FUNCTION_BLOCK XboxController
VAR_INPUT
END_VAR
VAR_OUTPUT
	
			XboxController				: 		FB_Xbox_Controller(NetID := '', iControllerNumber := 1);
			bIsConnected   				:  		ARRAY [1..2] OF BOOL;

			Start 						:       BOOL; 
			Reset 						:       BOOL;
			Button_A            		:       BOOL;
			Button_B                 	:       BOOL;
			Button_X             		:       BOOL;
			Button_Y                    :       BOOL;
			Dpad_U	                    :       BOOL;
			Dpad_D	                    :       BOOL;
			lBumper	                    :       BOOL;
			rBumper	                    :       BOOL;
			lTrigger                    :       LREAL;
			rTrigger                    :       LREAL;
			lStick_Y	                :       LREAL;
			lStick_X	                :       LREAL;
     		rStick_Y	                :       LREAL;
     		rStick_X	                :       LREAL;
			
END_VAR
VAR    
END_VAR

Cyclic();

METHOD clearScreenshot : BOOL
VAR_INPUT
	
bDpad_U 					: BOOL; 

END_VAR
END_METHOD

ACTION Cyclic:
XboxController.Cycle();
mapping(); 
init();
bIsConnected[1] := XboxController.P_Status.bConnected;
END_ACTION

METHOD Init
VAR_INPUT
END_VAR
END_METHOD

ACTION Mapping:




// Button Mapping
Start 				:= XboxController.P_Buttons.bStart;
Reset 				:= XboxController.P_Buttons.bBack;
Button_A 			:= XboxController.P_Buttons.bA_Button;
Button_B 			:= XboxController.P_Buttons.bB_Button;
Button_X 			:= XboxController.P_Buttons.bX_Button;
Button_Y 			:= XboxController.P_Buttons.bY_Button;
Dpad_U	 			:= XboxController.P_Buttons.DPad.bUp;
Dpad_D	 			:= XboxController.P_Buttons.DPad.bDown;
lBumper	 			:= XboxController.P_Buttons.bLeft_Shoulder;
rBumper	 			:= XboxController.P_Buttons.bRight_Shoulder;
lTrigger			:= XboxController.P_Left_Trigger;
rTrigger			:= XboxController.P_Right_Trigger;
lStick_Y			:= XboxController.P_Left_Joystick.fY;
lStick_X			:= XboxController.P_Left_Joystick.fX;
rStick_Y			:= XboxController.P_Right_Joystick.fY;
rStick_X			:= XboxController.P_Right_Joystick.fX;
END_ACTION

METHOD takeScreenshot : BOOL
VAR_INPUT
	
bDpad_D 				: BOOL ;

END_VAR
END_METHOD

END_FUNCTION_BLOCK

(* stored: Version 1.1.0.1, ProductVersion 3.1.4024.12
   POU XboxController: Id {90258775-ce06-40bc-98d6-66658f5c2f7b}, SpecialFunc None
   Folder Buttons: Id {b765c0d2-a1fa-47de-a83a-214fd5ccdffc}
   Method clearScreenshot: Id {8d5afaf2-b99a-41f7-9c02-692c817339db}
   Action Cyclic: Id {808b5749-855d-42fa-8193-f16ca32a0879}
   Method Init: Id {00fb4985-ae41-4cc3-9c5f-7e5a85b6bbf4}
   Action Mapping: Id {f5652c4a-9af9-40f9-9303-5deeb2d277c6}
   Method takeScreenshot: Id {f671d340-a431-47a9-bf30-27c82dc334e5} *)
